Yaskawa INFORM job: pipe_hz_cylinder_program.JBI

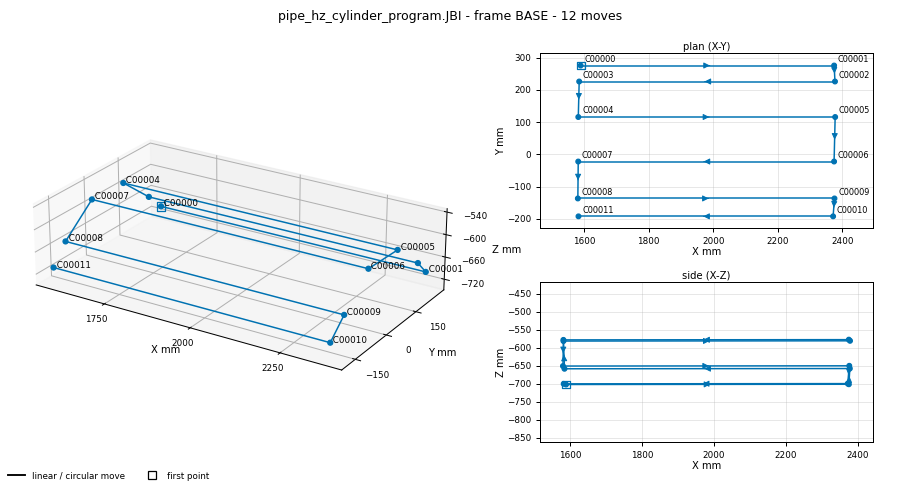
[picture p0: tool path of pipe_hz_cylinder_program.JBI in frame BASE, 12 of 15 moves have a stored position in this frame; points joined in program order, loops and branches not executed]
/JOB
//NAME pipe_hz_cylinder_program
//POS
///NPOS 12,0,12,0,0,0
///TOOL 0
///POSTYPE BASE
///RECTAN
///RCONF 0,0,0,0,0,0,0,0,0,0,0,0,0,0,0,0,0,0,0,0,0,0,0,0
C00000=1589.035645,275.284113,-702.216833,175.000000,-79.159246,-89.990945
C00001=2374.339912,275.284367,-701.570080,175.000000,-79.159246,-89.990945
C00002=2376.997086,225.791023,-657.905068,-175.000000,-51.554712,-89.962521
C00003=1584.668353,225.790767,-658.557607,-175.000000,-51.554712,-89.962521
C00004=1581.868901,115.789246,-581.593120,161.594609,-5.000000,5.000000
C00005=2377.557015,115.789504,-580.937815,161.594609,-5.000000,5.000000
C00006=2374.225642,-22.102220,-577.659258,-164.320940,-5.000000,-5.000000
C00007=1581.716896,-22.102477,-578.311944,-164.320940,-5.000000,-5.000000
C00008=1580.478965,-136.503484,-650.952767,175.000000,-49.148609,89.959214
C00009=2375.429085,-136.503227,-650.298070,175.000000,-49.148609,89.959214
C00010=2371.197292,-191.925281,-699.719381,175.000000,-77.889211,89.989893
C00011=1582.470658,-191.925537,-700.368952,180.000000,-60.000000,89.989893
///POSTYPE PULSE
///PULSE
EX00000=277504.0
///POSTYPE PULSE
///PULSE
EC00000=277504.0
EC00001=277504.0
EC00002=277504.0
EC00003=277504.0
EC00004=277504.0
EC00005=277504.0
EC00006=277504.0
EC00007=277504.0
EC00008=277504.0
EC00009=277504.0
EC00010=277504.0
EC00011=277504.0
//INST
///DATE 2023/08/15 13:18
///ATTR SC,RW,RJ
////FRAME BASE
///GROUP1 RB1,ST1
NOP
MOVJ P009 EX000 VJ=15.00
MOVJ C00000 EC00000 VJ=15.0
CALL JOB:SPYON
MOVL C00001 EC00001 V=150.0
MOVL C00002 EC00002 V=150.0
MOVL C00003 EC00003 V=150.0
MOVL C00004 EC00004 V=150.0
MOVL C00005 EC00005 V=150.0
MOVL C00006 EC00006 V=150.0
MOVL C00007 EC00007 V=150.0
MOVL C00008 EC00008 V=150.0
MOVL C00009 EC00009 V=150.0
MOVL C00010 EC00010 V=150.0
MOVL C00011 EC00011 V=150.0
CALL JOB:SPYOF
MOVJ P009 VJ=15.00
MOVL P009 EX00000 V=150.0
END
